PROGRAM MAIN
VAR
	input : BOOL;
	output : bool;
END_VAR

input := output;
Light();
Lamp();

END_PROGRAM

(* stored: Version 1.1.0.1, ProductVersion 3.1.4024.12
   POU MAIN: Id {b4d50afb-1b13-4589-a18b-61a811eeb4c7}, SpecialFunc None *)
